Staubli VAL3: loopReadForce.pgx

public program loopReadForce(num& x_nForceTorque[])
  local num l_nDetectValue[6]
begin

  //---------- 循环调用函数readDetectValue()读取传感器数值并转换成Force/Torque值 ----------

  //do

    //每4ms读取一次即可（否则会导致程序、任务卡死崩溃）
    //获取传感器的当前检测值
    call readDeteVal(l_nDetectValue)

    //计算传感器的Force/Torque数值并输出
    call calcForce(l_nDetectValue,x_nForceTorque)
    //delay(0.0)

  //until false

end
